% RSLogix 500 project PLC Level 2 Project 2.RSS, saved by version 8.30.00.16 %
PROJECT "UNTITLED"    % processor: Bul.1763 MicroLogix 1100 Series B %

PROGRAM FILES
  LAD 2 "MAIN"  3 rungs
  LAD 3 "IO CONFIG"  8 rungs
  LAD 4 "CTRL LOGIC"  10 rungs

DATA FILES
  O0 OUTPUT  4 elements
  I1 INPUT  6 elements
  S2 STATUS  66 elements
  B3 BINARY  2 elements
  T4 TIMER  1 elements
  C5 COUNTER  1 elements
  R6 CONTROL  1 elements
  N7 INTEGER  1 elements
  F8 FLOAT  1 elements

LADDER 2 "MAIN"
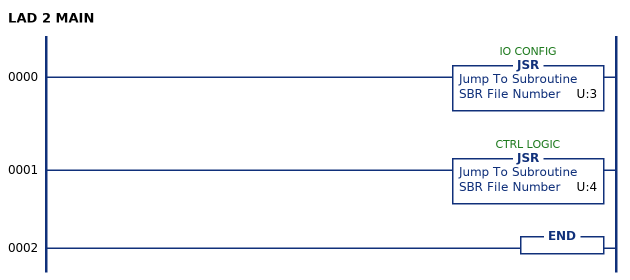
% Rung: 0 %
SOR JSR U:3 EOR
%   U:3  "IO CONFIG" %
% Rung: 1 %
SOR JSR U:4 EOR
%   U:4  "CTRL LOGIC" %
% Rung: 2 %
SOR END EOR

LADDER 3 "IO CONFIG"
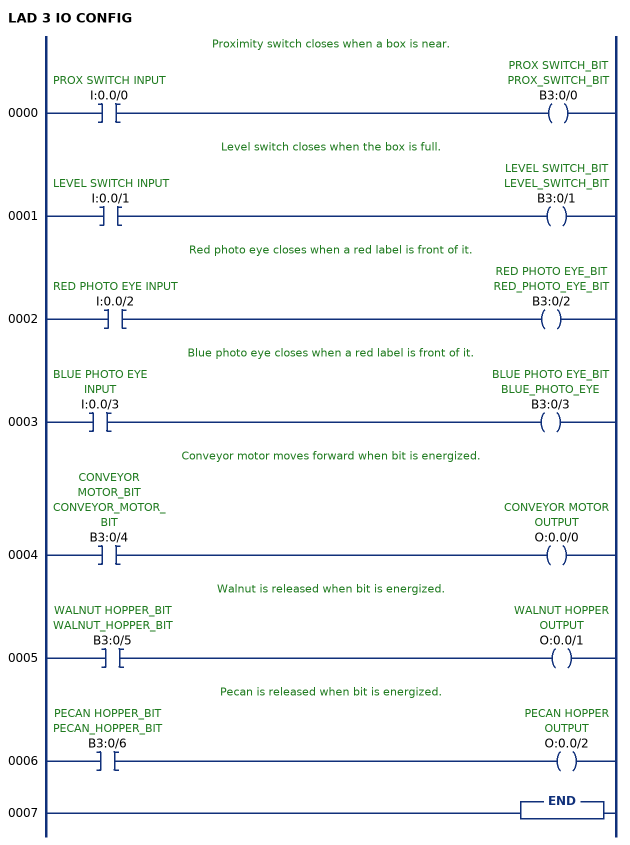
% Rung: 0 %
% Proximity switch closes when a box is near. %
SOR XIC I:0.0/0 OTE B3:0/0 EOR
%   I:0.0/0  "PROX SWITCH INPUT" %
%   B3:0/0  PROX_SWITCH_BIT  "PROX SWITCH_BIT" %
% Rung: 1 %
% Level switch closes when the box is full. %
SOR XIC I:0.0/1 OTE B3:0/1 EOR
%   I:0.0/1  "LEVEL SWITCH INPUT" %
%   B3:0/1  LEVEL_SWITCH_BIT  "LEVEL SWITCH_BIT" %
% Rung: 2 %
% Red photo eye closes when a red label is front of it. %
SOR XIC I:0.0/2 OTE B3:0/2 EOR
%   I:0.0/2  "RED PHOTO EYE INPUT" %
%   B3:0/2  RED_PHOTO_EYE_BIT  "RED PHOTO EYE_BIT" %
% Rung: 3 %
% Blue photo eye closes when a red label is front of it. %
SOR XIC I:0.0/3 OTE B3:0/3 EOR
%   I:0.0/3  "BLUE PHOTO EYE INPUT" %
%   B3:0/3  BLUE_PHOTO_EYE  "BLUE PHOTO EYE_BIT" %
% Rung: 4 %
% Conveyor motor moves forward when bit is energized. %
SOR XIC B3:0/4 OTE O:0.0/0 EOR
%   B3:0/4  CONVEYOR_MOTOR_BIT  "CONVEYOR MOTOR_BIT" %
%   O:0.0/0  "CONVEYOR MOTOR OUTPUT" %
% Rung: 5 %
% Walnut is released when bit is energized. %
SOR XIC B3:0/5 OTE O:0.0/1 EOR
%   B3:0/5  WALNUT_HOPPER_BIT  "WALNUT HOPPER_BIT" %
%   O:0.0/1  "WALNUT HOPPER OUTPUT" %
% Rung: 6 %
% Pecan is released when bit is energized. %
SOR XIC B3:0/6 OTE O:0.0/2 EOR
%   B3:0/6  PECAN_HOPPER_BIT  "PECAN HOPPER_BIT" %
%   O:0.0/2  "PECAN HOPPER OUTPUT" %
% Rung: 7 %
SOR END EOR

LADDER 4 "CTRL LOGIC"
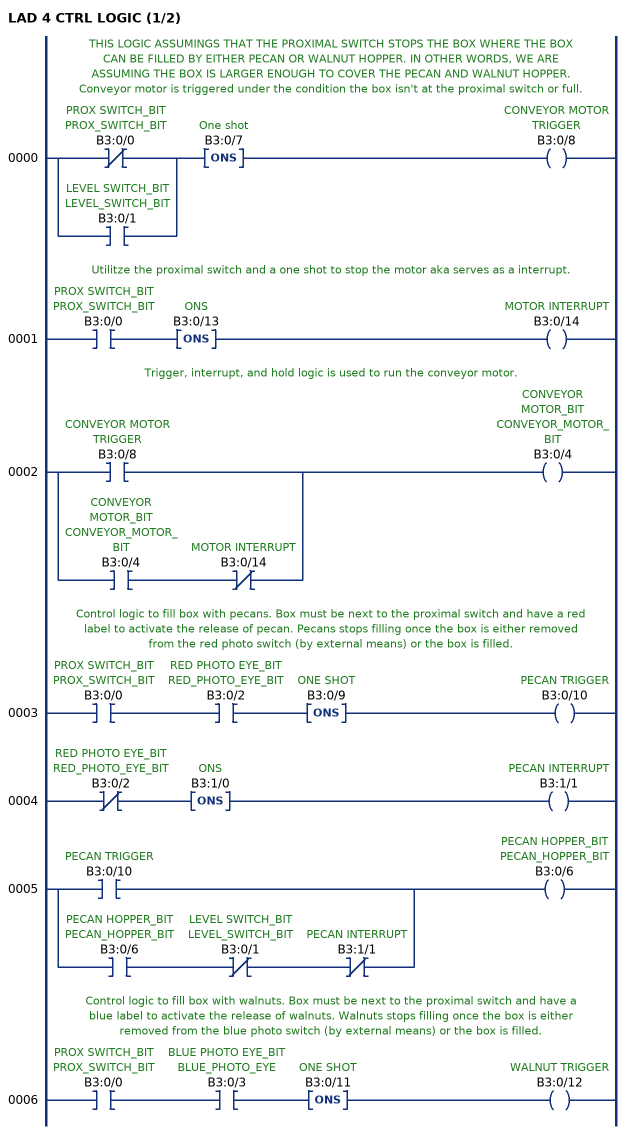
% Rung: 0 %
% THIS LOGIC ASSUMINGS THAT THE PROXIMAL SWITCH STOPS THE BOX WHERE THE BOX CAN BE FILLED BY EITHER PECAN OR WALNUT HOPPER. IN OTHER WORDS, WE ARE ASSUMING THE BOX IS LARGER ENOUGH TO COVER THE PECAN AND WALNUT HOPPER.
% Conveyor motor is triggered under the condition the box isn't at the proximal switch or full. %
SOR BST XIO B3:0/0 NXB XIC B3:0/1 BND ONS B3:0/7 OTE B3:0/8 EOR
%   B3:0/0  PROX_SWITCH_BIT  "PROX SWITCH_BIT" %
%   B3:0/1  LEVEL_SWITCH_BIT  "LEVEL SWITCH_BIT" %
%   B3:0/7  "One shot" %
%   B3:0/8  "CONVEYOR MOTOR TRIGGER" %
% Rung: 1 %
% Utilitze the proximal switch and a one shot to stop the motor aka serves as a interrupt. %
SOR XIC B3:0/0 ONS B3:0/13 OTE B3:0/14 EOR
%   B3:0/0  PROX_SWITCH_BIT  "PROX SWITCH_BIT" %
%   B3:0/13  "ONS" %
%   B3:0/14  "MOTOR INTERRUPT" %
% Rung: 2 %
% Trigger, interrupt, and hold logic is used to run the conveyor motor. %
SOR BST XIC B3:0/8 NXB XIC B3:0/4 XIO B3:0/14 BND OTE B3:0/4 EOR
%   B3:0/8  "CONVEYOR MOTOR TRIGGER" %
%   B3:0/4  CONVEYOR_MOTOR_BIT  "CONVEYOR MOTOR_BIT" %
%   B3:0/14  "MOTOR INTERRUPT" %
% Rung: 3 %
% Control logic to fill box with pecans. Box must be next to the proximal switch and have a red label to activate the release of pecan. Pecans stops filling once the box is either removed from the red photo switch (by external means) or the box is filled. %
SOR XIC B3:0/0 XIC B3:0/2 ONS B3:0/9 OTE B3:0/10 EOR
%   B3:0/0  PROX_SWITCH_BIT  "PROX SWITCH_BIT" %
%   B3:0/2  RED_PHOTO_EYE_BIT  "RED PHOTO EYE_BIT" %
%   B3:0/9  "ONE SHOT" %
%   B3:0/10  "PECAN TRIGGER" %
% Rung: 4 %
SOR XIO B3:0/2 ONS B3:1/0 OTE B3:1/1 EOR
%   B3:0/2  RED_PHOTO_EYE_BIT  "RED PHOTO EYE_BIT" %
%   B3:1/0  "ONS" %
%   B3:1/1  "PECAN INTERRUPT" %
% Rung: 5 %
SOR BST XIC B3:0/10 NXB XIC B3:0/6 XIO B3:0/1 XIO B3:1/1 BND OTE B3:0/6 EOR
%   B3:0/10  "PECAN TRIGGER" %
%   B3:0/6  PECAN_HOPPER_BIT  "PECAN HOPPER_BIT" %
%   B3:0/1  LEVEL_SWITCH_BIT  "LEVEL SWITCH_BIT" %
%   B3:1/1  "PECAN INTERRUPT" %
% Rung: 6 %
% Control logic to fill box with walnuts. Box must be next to the proximal switch and have a blue label to activate the release of walnuts. Walnuts stops filling once the box is either removed from the blue photo switch (by external means) or the box is filled. %
SOR XIC B3:0/0 XIC B3:0/3 ONS B3:0/11 OTE B3:0/12 EOR
%   B3:0/0  PROX_SWITCH_BIT  "PROX SWITCH_BIT" %
%   B3:0/3  BLUE_PHOTO_EYE  "BLUE PHOTO EYE_BIT" %
%   B3:0/11  "ONE SHOT" %
%   B3:0/12  "WALNUT TRIGGER" %

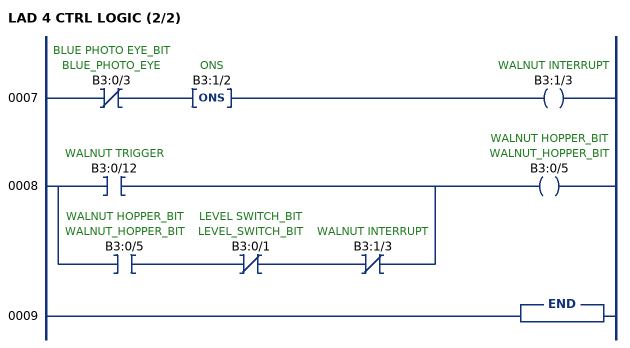
% Rung: 7 %
SOR XIO B3:0/3 ONS B3:1/2 OTE B3:1/3 EOR
%   B3:0/3  BLUE_PHOTO_EYE  "BLUE PHOTO EYE_BIT" %
%   B3:1/2  "ONS" %
%   B3:1/3  "WALNUT INTERRUPT" %
% Rung: 8 %
SOR BST XIC B3:0/12 NXB XIC B3:0/5 XIO B3:0/1 XIO B3:1/3 BND OTE B3:0/5 EOR
%   B3:0/12  "WALNUT TRIGGER" %
%   B3:0/5  WALNUT_HOPPER_BIT  "WALNUT HOPPER_BIT" %
%   B3:0/1  LEVEL_SWITCH_BIT  "LEVEL SWITCH_BIT" %
%   B3:1/3  "WALNUT INTERRUPT" %
% Rung: 9 %
SOR END EOR
